{attribute addProperty BoxType "EK1960-2600-0021"}
{attribute addProperty Id "FSoE_CommandUSINT811FSOUT_Module_1_Channel_1_Output_X5_1BIT10.1251FSOUT_Module_1_Channel_2_Output_X5_2BIT10.1252FSOUT_Module_1_Channel_3_Output_X5_3BIT10.1253FSOUT_Module_1_Channel_4_Output_X5_4BIT10.1254FSOUT_Module_1_ErrAckBIT10.1251FSOUT_Module_2_Channel_1_Output_X5_5BIT10.1251FSOUT_Module_2_Channel_2_Output_X5_6BIT10.1252FSOUT_Module_2_Channel_3_Output_X5_7BIT10.1253FSOUT_Module_2_Channel_4_Output_X5_8BIT10.1254FSOUT_Module_2_ErrAckBIT10.1251FSOUT_Module_3_Channel_1_Output_X7_1BIT10.1251FSOUT_Module_3_Channel_2_Output_X7_2BIT10.1252FSOUT_Module_3_Channel_3_Output_X7_3BIT10.1253FSOUT_Module_3_Channel_4_Output_X7_4BIT10.1254FSOUT_Module_3_ErrAckBIT10.1251FSOUT_Module_4_Channel_1_Output_X7_5BIT10.1251FSoE_CRC_000UINT1623FSOUT_Module_4_Channel_2_Output_X7_6BIT10.1252FSOUT_Module_4_Channel_3_Output_X7_7BIT10.1253FSOUT_Module_4_Channel_4_Output_X7_8BIT10.1254FSOUT_Module_4_ErrAckBIT10.1251FSOUT_Module_5_Channel_1_Output_X9_1BIT10.1251FSOUT_Module_5_Channel_2_Output_X9_2BIT10.1252FSOUT_Module_5_Channel_3_Output_X9_3BIT10.1253FSOUT_Module_5_Channel_4_Output_X9_4BIT10.1254FSOUT_Module_5_ErrAckBIT10.1251FSOUT_Module_6_Channel_1_Output_X9_5BIT10.1251FSOUT_Module_6_Channel_2_Output_X9_6BIT10.1252FSOUT_Module_6_Channel_3_Output_X9_7BIT10.1253FSOUT_Module_6_Channel_4_Output_X9_8BIT10.1254FSOUT_Module_6_ErrAckBIT10.1251FSOUT_Relais_Module_Channel_1_Output_X4_1_X4_5BIT10.1251FSOUT_Relais_Module_Channel_2_Output_X4_2_X4_6BIT10.1252FSoE_CRC_001UINT1624FSOUT_Relais_Module_Channel_3_Output_X4_3_X4_7BIT10.1253FSOUT_Relais_Module_Channel_4_Output_X4_4_X4_8BIT10.1254FSOUT_Relais_Module_ErrAckBIT10.1251FSIN_Module_1_ErrAckBIT10.1251FSIN_Module_2_ErrAckBIT10.1251FSIN_Module_3_ErrAckBIT10.1251FSIN_Module_4_ErrAckBIT10.1251FSIN_Module_5_ErrAckBIT10.1251FSIN_Module_6_ErrAckBIT10.1251FSIN_Module_7_ErrAckBIT10.1251FSIN_Module_8_ErrAckBIT10.1251FSIN_Module_9_Err_Ack_1BIT10.1251FSIN_Module_9_Err_Ack_2BIT10.1252FSIN_Module_10_Err_Ack_1BIT10.1251FSIN_Module_10_Err_Ack_2BIT10.1252FSoE_CRC_002UINT1625FSoE_Connection_IDUINT1622"}
{attribute addProperty CRC "2667934578"}
{attribute addProperty SizeInBites "120"}
{attribute addProperty SizeInBytes "15"}
TYPE FSOE_9F057372 :
STRUCT
	{attribute addProperty Name "FSoE_Command"}
	FSoE_Command : USINT;
	{attribute addProperty Name "FSOUT_Module_1_Channel_1_Output_X5_1"}
	FSOUT_Module_1_Channel_1_Output_X5_1 : BOOL;
	{attribute addProperty Name "FSOUT_Module_1_Channel_2_Output_X5_2"}
	FSOUT_Module_1_Channel_2_Output_X5_2 : BOOL;
	{attribute addProperty Name "FSOUT_Module_1_Channel_3_Output_X5_3"}
	FSOUT_Module_1_Channel_3_Output_X5_3 : BOOL;
	{attribute addProperty Name "FSOUT_Module_1_Channel_4_Output_X5_4"}
	FSOUT_Module_1_Channel_4_Output_X5_4 : BOOL;
	{attribute addProperty Name "FSOUT_Module_1_ErrAck"}
	FSOUT_Module_1_ErrAck : BOOL;
	{attribute addProperty Name "FSOUT_Module_2_Channel_1_Output_X5_5"}
	FSOUT_Module_2_Channel_1_Output_X5_5 : BOOL;
	{attribute addProperty Name "FSOUT_Module_2_Channel_2_Output_X5_6"}
	FSOUT_Module_2_Channel_2_Output_X5_6 : BOOL;
	{attribute addProperty Name "FSOUT_Module_2_Channel_3_Output_X5_7"}
	FSOUT_Module_2_Channel_3_Output_X5_7 : BOOL;
	{attribute addProperty Name "FSOUT_Module_2_Channel_4_Output_X5_8"}
	FSOUT_Module_2_Channel_4_Output_X5_8 : BOOL;
	{attribute addProperty Name "FSOUT_Module_2_ErrAck"}
	FSOUT_Module_2_ErrAck : BOOL;
	{attribute addProperty Name "FSOUT_Module_3_Channel_1_Output_X7_1"}
	FSOUT_Module_3_Channel_1_Output_X7_1 : BOOL;
	{attribute addProperty Name "FSOUT_Module_3_Channel_2_Output_X7_2"}
	FSOUT_Module_3_Channel_2_Output_X7_2 : BOOL;
	{attribute addProperty Name "FSOUT_Module_3_Channel_3_Output_X7_3"}
	FSOUT_Module_3_Channel_3_Output_X7_3 : BOOL;
	{attribute addProperty Name "FSOUT_Module_3_Channel_4_Output_X7_4"}
	FSOUT_Module_3_Channel_4_Output_X7_4 : BOOL;
	{attribute addProperty Name "FSOUT_Module_3_ErrAck"}
	FSOUT_Module_3_ErrAck : BOOL;
	{attribute addProperty Name "FSOUT_Module_4_Channel_1_Output_X7_5"}
	FSOUT_Module_4_Channel_1_Output_X7_5 : BOOL;
	{attribute addProperty Name "FSoE_CRC_000"}
	FSoE_CRC_000 : UINT;
	{attribute addProperty Name "FSOUT_Module_4_Channel_2_Output_X7_6"}
	FSOUT_Module_4_Channel_2_Output_X7_6 : BOOL;
	{attribute addProperty Name "FSOUT_Module_4_Channel_3_Output_X7_7"}
	FSOUT_Module_4_Channel_3_Output_X7_7 : BOOL;
	{attribute addProperty Name "FSOUT_Module_4_Channel_4_Output_X7_8"}
	FSOUT_Module_4_Channel_4_Output_X7_8 : BOOL;
	{attribute addProperty Name "FSOUT_Module_4_ErrAck"}
	FSOUT_Module_4_ErrAck : BOOL;
	{attribute addProperty Name "FSOUT_Module_5_Channel_1_Output_X9_1"}
	FSOUT_Module_5_Channel_1_Output_X9_1 : BOOL;
	{attribute addProperty Name "FSOUT_Module_5_Channel_2_Output_X9_2"}
	FSOUT_Module_5_Channel_2_Output_X9_2 : BOOL;
	{attribute addProperty Name "FSOUT_Module_5_Channel_3_Output_X9_3"}
	FSOUT_Module_5_Channel_3_Output_X9_3 : BOOL;
	{attribute addProperty Name "FSOUT_Module_5_Channel_4_Output_X9_4"}
	FSOUT_Module_5_Channel_4_Output_X9_4 : BOOL;
	{attribute addProperty Name "FSOUT_Module_5_ErrAck"}
	FSOUT_Module_5_ErrAck : BOOL;
	{attribute addProperty Name "FSOUT_Module_6_Channel_1_Output_X9_5"}
	FSOUT_Module_6_Channel_1_Output_X9_5 : BOOL;
	{attribute addProperty Name "FSOUT_Module_6_Channel_2_Output_X9_6"}
	FSOUT_Module_6_Channel_2_Output_X9_6 : BOOL;
	{attribute addProperty Name "FSOUT_Module_6_Channel_3_Output_X9_7"}
	FSOUT_Module_6_Channel_3_Output_X9_7 : BOOL;
	{attribute addProperty Name "FSOUT_Module_6_Channel_4_Output_X9_8"}
	FSOUT_Module_6_Channel_4_Output_X9_8 : BOOL;
	{attribute addProperty Name "FSOUT_Module_6_ErrAck"}
	FSOUT_Module_6_ErrAck : BOOL;
	{attribute addProperty Name "FSOUT_Relais_Module_Channel_1_Output_X4_1_X4_5"}
	FSOUT_Relais_Module_Channel_1_Output_X4_1_X4_5 : BOOL;
	{attribute addProperty Name "FSOUT_Relais_Module_Channel_2_Output_X4_2_X4_6"}
	FSOUT_Relais_Module_Channel_2_Output_X4_2_X4_6 : BOOL;
	{attribute addProperty Name "FSoE_CRC_001"}
	FSoE_CRC_001 : UINT;
	{attribute addProperty Name "FSOUT_Relais_Module_Channel_3_Output_X4_3_X4_7"}
	FSOUT_Relais_Module_Channel_3_Output_X4_3_X4_7 : BOOL;
	{attribute addProperty Name "FSOUT_Relais_Module_Channel_4_Output_X4_4_X4_8"}
	FSOUT_Relais_Module_Channel_4_Output_X4_4_X4_8 : BOOL;
	{attribute addProperty Name "FSOUT_Relais_Module_ErrAck"}
	FSOUT_Relais_Module_ErrAck : BOOL;
	{attribute addProperty Name "FSIN_Module_1_ErrAck"}
	FSIN_Module_1_ErrAck : BOOL;
	{attribute addProperty Name "FSIN_Module_2_ErrAck"}
	FSIN_Module_2_ErrAck : BOOL;
	{attribute addProperty Name "FSIN_Module_3_ErrAck"}
	FSIN_Module_3_ErrAck : BOOL;
	{attribute addProperty Name "FSIN_Module_4_ErrAck"}
	FSIN_Module_4_ErrAck : BOOL;
	{attribute addProperty Name "FSIN_Module_5_ErrAck"}
	FSIN_Module_5_ErrAck : BOOL;
	{attribute addProperty Name "FSIN_Module_6_ErrAck"}
	FSIN_Module_6_ErrAck : BOOL;
	{attribute addProperty Name "FSIN_Module_7_ErrAck"}
	FSIN_Module_7_ErrAck : BOOL;
	{attribute addProperty Name "FSIN_Module_8_ErrAck"}
	FSIN_Module_8_ErrAck : BOOL;
	{attribute addProperty Name "FSIN_Module_9_Err_Ack_1"}
	FSIN_Module_9_Err_Ack_1 : BOOL;
	{attribute addProperty Name "FSIN_Module_9_Err_Ack_2"}
	FSIN_Module_9_Err_Ack_2 : BOOL;
	{attribute addProperty Name "FSIN_Module_10_Err_Ack_1"}
	FSIN_Module_10_Err_Ack_1 : BOOL;
	{attribute addProperty Name "FSIN_Module_10_Err_Ack_2"}
	FSIN_Module_10_Err_Ack_2 : BOOL;
	{attribute 'hide'}
	reserve_1 : BOOL;
	{attribute addProperty Name "FSoE_CRC_002"}
	FSoE_CRC_002 : UINT;
	{attribute addProperty Name "FSoE_Connection_ID"}
	FSoE_Connection_ID : UINT;
END_STRUCT
END_TYPE

(* stored: Version 1.2.0.0, ProductVersion 3.1.4024.9
   DUT FSOE_9F057372: Id {2cc0c04c-8d03-47dc-b352-ba2efb2485f8} *)
